// Mitsubishi GX Works2 project: IND_Plastificiranje_Termin6   PLC: FX3S

// task Task_01 (event TRUE, interval 0, priority 31): POU_01

PROGRAM POU_01
VAR
  zona_uslova_1 : zona_uslova;
  START_Taster : BOOL;
  STOP_taster : BOOL;
  Pokreni_proces_taster : BOOL;
  Termostat : BOOL;
  ukljucen_sistem : BOOL;
  prelazak0_1 : BOOL;
  prelazak1_2 : BOOL;
  prelazak2_3 : BOOL;
  prelazak3_4 : BOOL;
  prelazak4_0 : BOOL;
  zona_prelaza_1 : zona_prelaza;
  en_cyc : BOOL;
  step_by_step : BOOL;
  next_step : BOOL;
  trenutno_stanje : INT;
  tr_st0 : BOOL;
  tr_st1 : BOOL;
  tr_st2 : BOOL;
  tr_st3 : BOOL;
  tr_st4 : BOOL;
  zona_izvrsenja_1 : zona_izvrsenja;
  man_grejac : BOOL;
  man_ventilator : BOOL;
  man_svetlo : BOOL;
  Grejac : BOOL;
  Ventilator : BOOL;
  Svetlo : BOOL;
END_VAR
(* structured ladder/FBD written out as ST: instructions are called as NAME(EN, inputs, outputs); _pN, _eN, _tN stand for wires *)
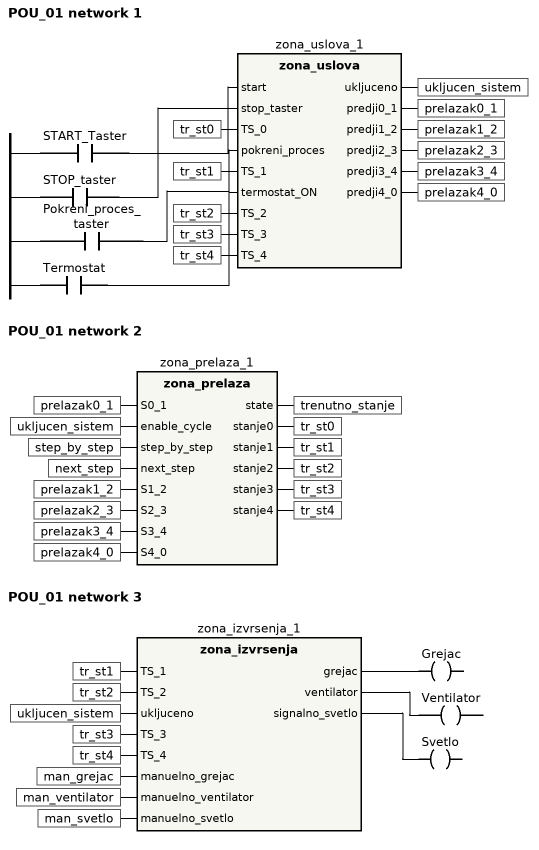
(* network 1 *)
zona_uslova_1(start := START_Taster, stop_taster := STOP_taster, TS_0 := tr_st0, pokreni_proces := Pokreni_proces_taster, TS_1 := tr_st1, termostat_ON := Termostat, TS_2 := tr_st2, TS_3 := tr_st3, TS_4 := tr_st4, ukljuceno => ukljucen_sistem, predji0_1 => prelazak0_1, predji1_2 => prelazak1_2, predji2_3 => prelazak2_3, predji3_4 => prelazak3_4, predji4_0 => prelazak4_0);
(* network 2 *)
zona_prelaza_1(S0_1 := prelazak0_1, enable_cycle := ukljucen_sistem, step_by_step := step_by_step, next_step := next_step, S1_2 := prelazak1_2, S2_3 := prelazak2_3, S3_4 := prelazak3_4, S4_0 := prelazak4_0, state => trenutno_stanje, stanje0 => tr_st0, stanje1 => tr_st1, stanje2 => tr_st2, stanje3 => tr_st3, stanje4 => tr_st4);
(* network 3 *)
zona_izvrsenja_1(TS_1 := tr_st1, TS_2 := tr_st2, ukljuceno := ukljucen_sistem, TS_3 := tr_st3, TS_4 := tr_st4, manuelno_grejac := man_grejac, manuelno_ventilator := man_ventilator, manuelno_svetlo := man_svetlo);
Grejac := zona_izvrsenja_1.grejac;
Ventilator := zona_izvrsenja_1.ventilator;
Svetlo := zona_izvrsenja_1.signalno_svetlo;
END_PROGRAM

FUNCTION_BLOCK zona_prelaza
VAR_OUTPUT
  state : INT;
END_VAR
VAR
  jednako : ARRAY [0..2] OF BOOL;
END_VAR
VAR_INPUT
  S0_1 : BOOL;
  enable_cycle : BOOL;
  step_by_step : BOOL;
  next_step : BOOL;
  S1_2 : BOOL;
  S2_3 : BOOL;
  S3_4 : BOOL;
  S4_0 : BOOL;
END_VAR
VAR_OUTPUT
  stanje0 : BOOL;
  stanje1 : BOOL;
  stanje2 : BOOL;
  stanje3 : BOOL;
  stanje4 : BOOL;
END_VAR
(* structured ladder/FBD written out as ST: instructions are called as NAME(EN, inputs, outputs); _pN, _eN, _tN stand for wires *)
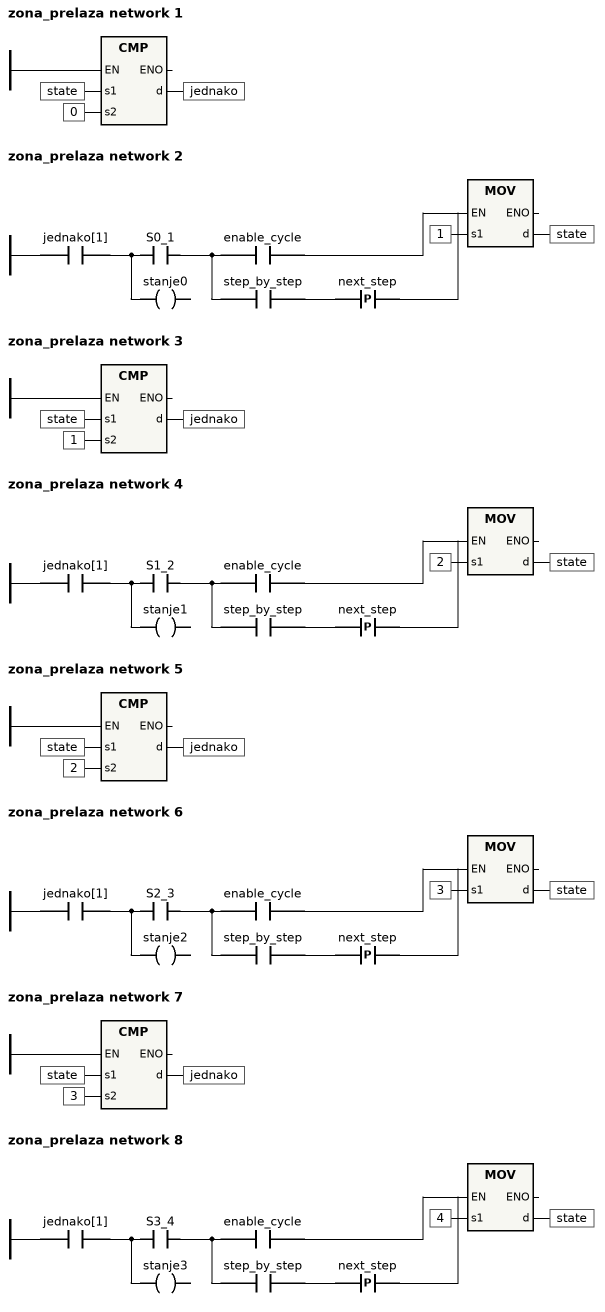
(* network 1 *)
CMP(TRUE, state, 0, jednako);
(* network 2 *)
_p1 := jednako[1] AND S0_1;
MOV((_p1 AND enable_cycle) OR (_p1 AND step_by_step AND LDP(TRUE, next_step)), 1, state);
stanje0 := jednako[1];
(* network 3 *)
CMP(TRUE, state, 1, jednako);
(* network 4 *)
_p1 := jednako[1] AND S1_2;
MOV((_p1 AND enable_cycle) OR (_p1 AND step_by_step AND LDP(TRUE, next_step)), 2, state);
stanje1 := jednako[1];
(* network 5 *)
CMP(TRUE, state, 2, jednako);
(* network 6 *)
_p1 := jednako[1] AND S2_3;
MOV((_p1 AND enable_cycle) OR (_p1 AND step_by_step AND LDP(TRUE, next_step)), 3, state);
stanje2 := jednako[1];
(* network 7 *)
CMP(TRUE, state, 3, jednako);
(* network 8 *)
_p1 := jednako[1] AND S3_4;
MOV((_p1 AND enable_cycle) OR (_p1 AND step_by_step AND LDP(TRUE, next_step)), 4, state);
stanje3 := jednako[1];
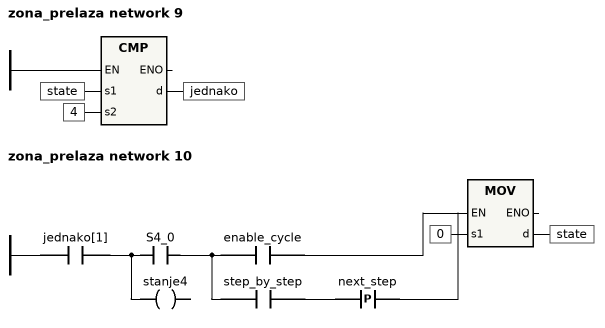
(* network 9 *)
CMP(TRUE, state, 4, jednako);
(* network 10 *)
_p1 := jednako[1] AND S4_0;
MOV((_p1 AND enable_cycle) OR (_p1 AND step_by_step AND LDP(TRUE, next_step)), 0, state);
stanje4 := jednako[1];
END_FUNCTION_BLOCK

FUNCTION_BLOCK zona_uslova
VAR_INPUT
  start : BOOL;
  stop_taster : BOOL;
END_VAR
VAR_OUTPUT
  ukljuceno : BOOL;
END_VAR
VAR_INPUT
  TS_0 : BOOL;
  pokreni_proces : BOOL;
END_VAR
VAR_OUTPUT
  predji0_1 : BOOL;
END_VAR
VAR_INPUT
  TS_1 : BOOL;
  termostat_ON : BOOL;
END_VAR
VAR_OUTPUT
  predji1_2 : BOOL;
END_VAR
VAR_INPUT
  TS_2 : BOOL;
END_VAR
VAR
  TON_1 : TON;
  vreme_tajmera1 : TIME;
END_VAR
VAR_OUTPUT
  predji2_3 : BOOL;
END_VAR
VAR_INPUT
  TS_3 : BOOL;
END_VAR
VAR
  TON_2 : TON;
  vreme_tajmera2 : TIME;
END_VAR
VAR_OUTPUT
  predji3_4 : BOOL;
END_VAR
VAR_INPUT
  TS_4 : BOOL;
END_VAR
VAR
  TON_3 : TON;
  vreme_tajmera3 : TIME;
END_VAR
VAR_OUTPUT
  predji4_0 : BOOL;
END_VAR
(* structured ladder/FBD written out as ST: instructions are called as NAME(EN, inputs, outputs); _pN, _eN, _tN stand for wires *)
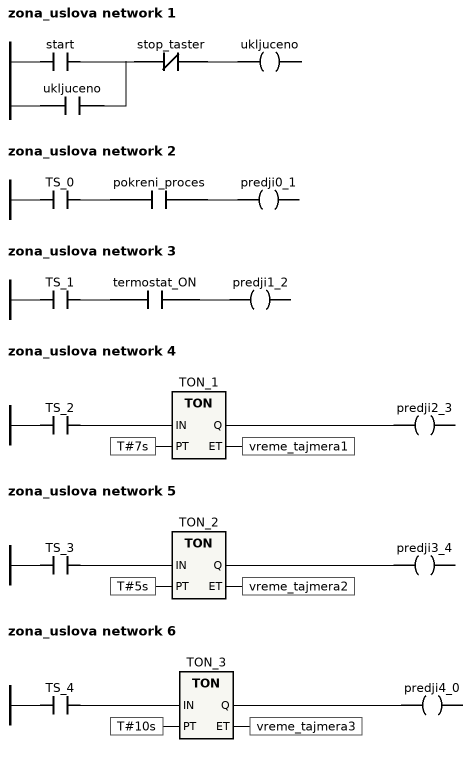
(* network 1 *)
ukljuceno := (start OR ukljuceno) AND NOT stop_taster;
(* network 2 *)
predji0_1 := TS_0 AND pokreni_proces;
(* network 3 *)
predji1_2 := TS_1 AND termostat_ON;
(* network 4 *)
TON_1(IN := TS_2, PT := T#7s, ET => vreme_tajmera1);
predji2_3 := TON_1.Q;
(* network 5 *)
TON_2(IN := TS_3, PT := T#5s, ET => vreme_tajmera2);
predji3_4 := TON_2.Q;
(* network 6 *)
TON_3(IN := TS_4, PT := T#10s, ET => vreme_tajmera3);
predji4_0 := TON_3.Q;
END_FUNCTION_BLOCK

FUNCTION_BLOCK zona_izvrsenja
VAR_INPUT
  TS_1 : BOOL;
  TS_2 : BOOL;
  ukljuceno : BOOL;
END_VAR
VAR_OUTPUT
  grejac : BOOL;
END_VAR
VAR_INPUT
  TS_3 : BOOL;
END_VAR
VAR_OUTPUT
  ventilator : BOOL;
END_VAR
VAR_INPUT
  TS_4 : BOOL;
END_VAR
VAR_OUTPUT
  signalno_svetlo : BOOL;
END_VAR
VAR_INPUT
  manuelno_grejac : BOOL;
  manuelno_ventilator : BOOL;
  manuelno_svetlo : BOOL;
END_VAR
(* structured ladder/FBD written out as ST: instructions are called as NAME(EN, inputs, outputs); _pN, _eN, _tN stand for wires *)
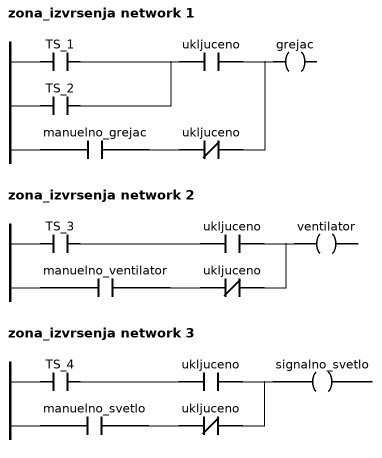
(* network 1 *)
grejac := ((TS_1 OR TS_2) AND ukljuceno) OR (manuelno_grejac AND NOT ukljuceno);
(* network 2 *)
ventilator := (TS_3 AND ukljuceno) OR (manuelno_ventilator AND NOT ukljuceno);
(* network 3 *)
signalno_svetlo := (TS_4 AND ukljuceno) OR (manuelno_svetlo AND NOT ukljuceno);
END_FUNCTION_BLOCK
